// LS Electric XG5000 project: 커스텀통신시도1
// PLC LSPLC

PROGRAM NewProgram (task: 스캔 프로그램)

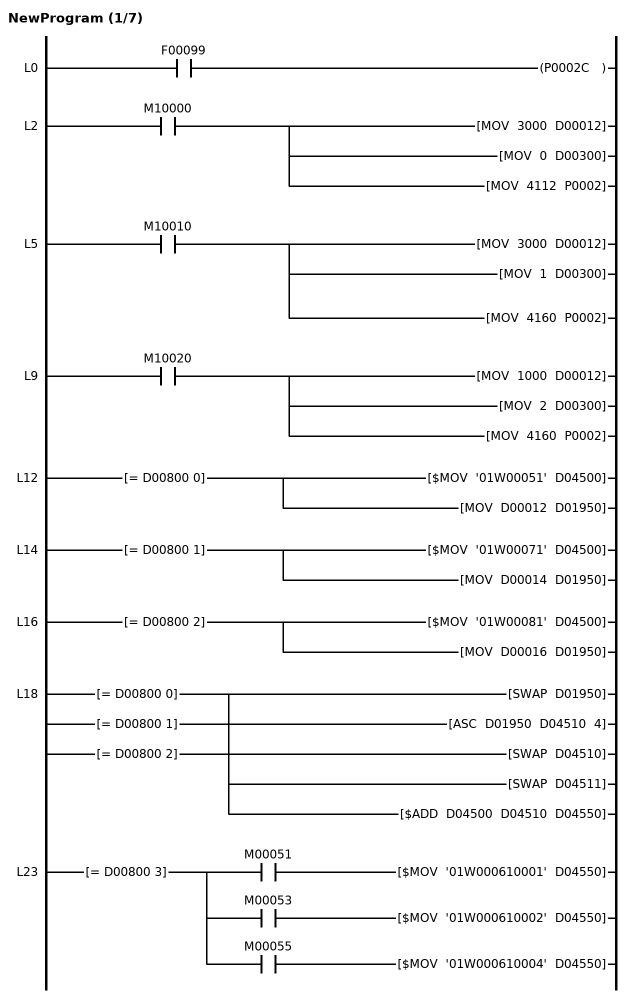
; L0
LOAD      F00099
OUT       P0002C
; L2
LOAD      M10000
MOV       3000 D00012
MOV       0 D00300
MOV       4112 P0002
; L5
LOAD      M10010
MOV       3000 D00012
MOV       1 D00300
MOV       4160 P0002
; L9
LOAD      M10020
MOV       1000 D00012
MOV       2 D00300
MOV       4160 P0002
; L12
LOAD=     D00800 0
$MOV      '01W00051' D04500
MOV       D00012 D01950
; L14
LOAD=     D00800 1
$MOV      '01W00071' D04500
MOV       D00014 D01950
; L16
LOAD=     D00800 2
$MOV      '01W00081' D04500
MOV       D00016 D01950
; L18
LOAD=     D00800 0
OR=       D00800 1
OR=       D00800 2
SWAP      D01950
ASC       D01950 D04510 4
SWAP      D04510
SWAP      D04511
$ADD      D04500 D04510 D04550
; L23
LOAD=     D00800 3
MPUSH
AND       M00051
$MOV      '01W000610001' D04550
MLOAD
AND       M00053
$MOV      '01W000610002' D04550
MPOP
AND       M00055
$MOV      '01W000610004' D04550

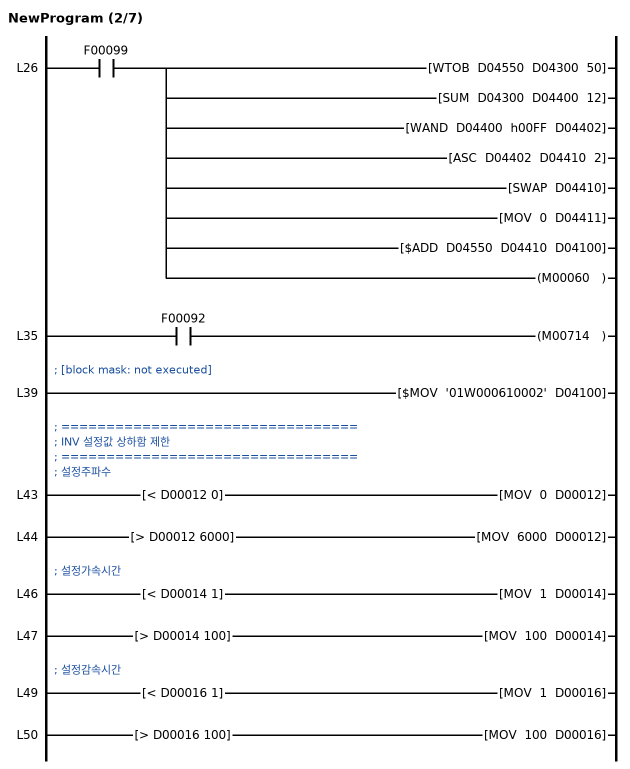
; L26
LOAD      F00099
WTOB      D04550 D04300 50
SUM       D04300 D04400 12
WAND      D04400 h00FF D04402
ASC       D04402 D04410 2
SWAP      D04410
MOV       0 D04411
$ADD      D04550 D04410 D04100
OUT       M00060
; L35
LOAD      F00092
OUT       M00714
; L39 (block mask: not executed)
$MOV      '01W000610002' D04100
// =================================
//    INV 설정값 상하함 제한
// =================================
// 설정주파수
; L43
LOAD<     D00012 0
MOV       0 D00012
; L44
LOAD>     D00012 6000
MOV       6000 D00012
// 설정가속시간
; L46
LOAD<     D00014 1
MOV       1 D00014
; L47
LOAD>     D00014 100
MOV       100 D00014
// 설정감속시간
; L49
LOAD<     D00016 1
MOV       1 D00016
; L50
LOAD>     D00016 100
MOV       100 D00016

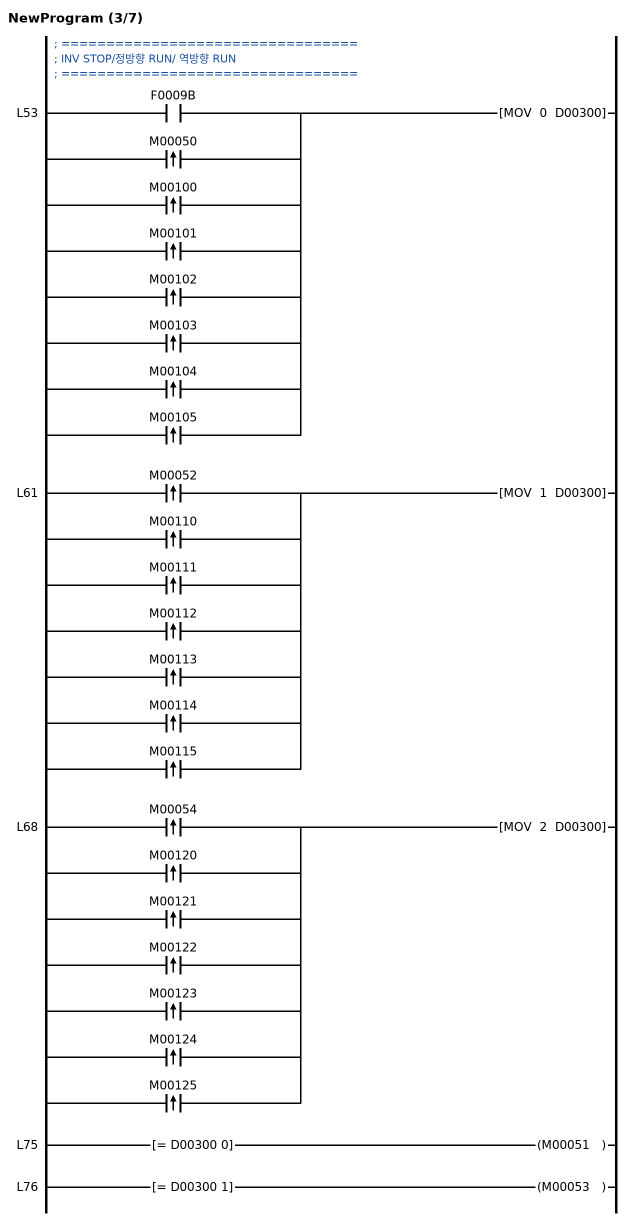
// =================================
//    INV STOP/정방향 RUN/ 역방향 RUN
// =================================
; L53
LOAD      F0009B
ORP       M00050
ORP       M00100
ORP       M00101
ORP       M00102
ORP       M00103
ORP       M00104
ORP       M00105
MOV       0 D00300
; L61
LOADP     M00052
ORP       M00110
ORP       M00111
ORP       M00112
ORP       M00113
ORP       M00114
ORP       M00115
MOV       1 D00300
; L68
LOADP     M00054
ORP       M00120
ORP       M00121
ORP       M00122
ORP       M00123
ORP       M00124
ORP       M00125
MOV       2 D00300
; L75
LOAD=     D00300 0
OUT       M00051
; L76
LOAD=     D00300 1
OUT       M00053

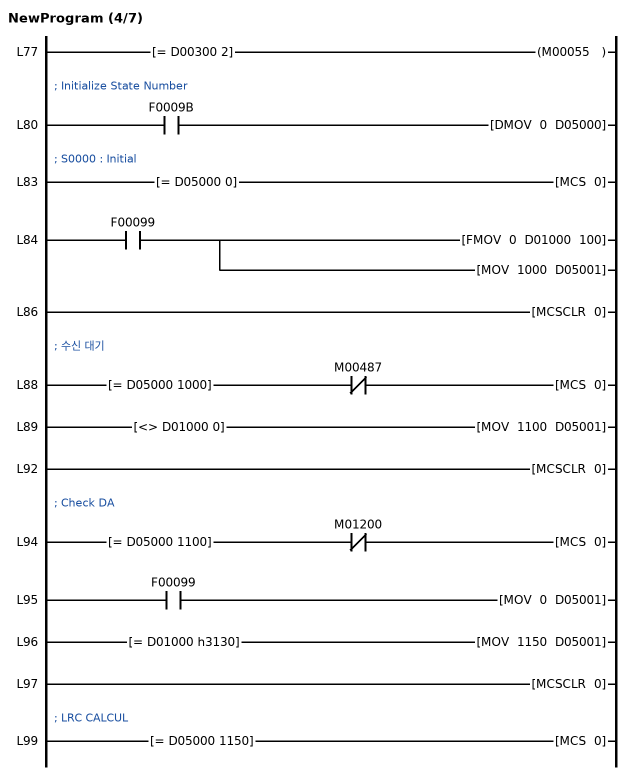
; L77
LOAD=     D00300 2
OUT       M00055
// Initialize State Number
; L80
LOAD      F0009B
DMOV      0 D05000
// S0000 : Initial
; L83
LOAD=     D05000 0
MCS       0
; L84
LOAD      F00099
FMOV      0 D01000 100
MOV       1000 D05001
; L86
MCSCLR    0
// 수신 대기
; L88
LOAD=     D05000 1000
AND NOT   M00487
MCS       0
; L89
LOAD<>    D01000 0
MOV       1100 D05001
; L92
MCSCLR    0
// Check DA
; L94
LOAD=     D05000 1100
AND NOT   M01200
MCS       0
; L95
LOAD      F00099
MOV       0 D05001
; L96
LOAD=     D01000 h3130
MOV       1150 D05001
; L97
MCSCLR    0
// LRC CALCUL
; L99
LOAD=     D05000 1150
MCS       0

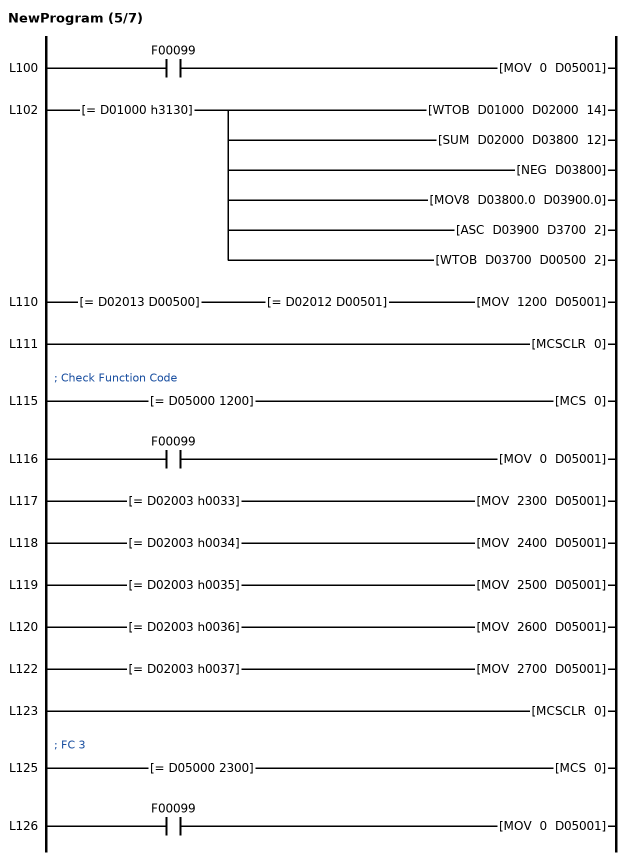
; L100
LOAD      F00099
MOV       0 D05001
; L102
LOAD=     D01000 h3130
WTOB      D01000 D02000 14
SUM       D02000 D03800 12
NEG       D03800
MOV8      D03800.0 D03900.0
ASC       D03900 D3700 2
WTOB      D03700 D00500 2
; L110
LOAD=     D02013 D00500
AND=      D02012 D00501
MOV       1200 D05001
; L111
MCSCLR    0
// Check Function Code
; L115
LOAD=     D05000 1200
MCS       0
; L116
LOAD      F00099
MOV       0 D05001
; L117
LOAD=     D02003 h0033
MOV       2300 D05001
; L118
LOAD=     D02003 h0034
MOV       2400 D05001
; L119
LOAD=     D02003 h0035
MOV       2500 D05001
; L120
LOAD=     D02003 h0036
MOV       2600 D05001
; L122
LOAD=     D02003 h0037
MOV       2700 D05001
; L123
MCSCLR    0
// FC 3
; L125
LOAD=     D05000 2300
MCS       0
; L126
LOAD      F00099
MOV       0 D05001

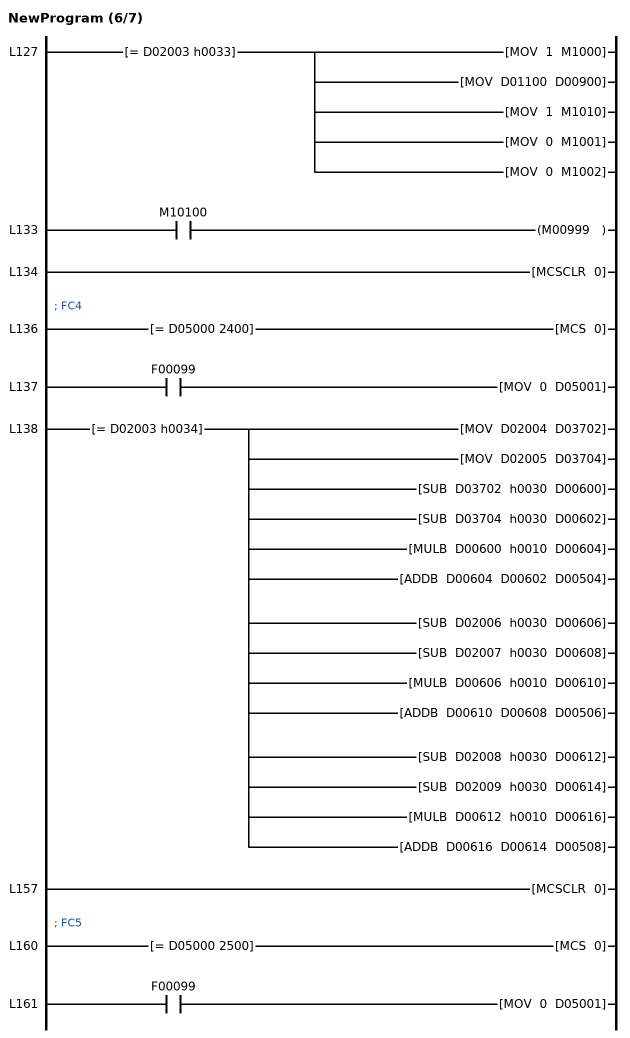
; L127
LOAD=     D02003 h0033
MOV       1 M1000
MOV       D01100 D00900
MOV       1 M1010
MOV       0 M1001
MOV       0 M1002
; L133
LOAD      M10100
OUT       M00999
; L134
MCSCLR    0
// FC4
; L136
LOAD=     D05000 2400
MCS       0
; L137
LOAD      F00099
MOV       0 D05001
; L138
LOAD=     D02003 h0034
MOV       D02004 D03702
MOV       D02005 D03704
SUB       D03702 h0030 D00600
SUB       D03704 h0030 D00602
MULB      D00600 h0010 D00604
ADDB      D00604 D00602 D00504
SUB       D02006 h0030 D00606
SUB       D02007 h0030 D00608
MULB      D00606 h0010 D00610
ADDB      D00610 D00608 D00506
SUB       D02008 h0030 D00612
SUB       D02009 h0030 D00614
MULB      D00612 h0010 D00616
ADDB      D00616 D00614 D00508
; L157
MCSCLR    0
// FC5
; L160
LOAD=     D05000 2500
MCS       0
; L161
LOAD      F00099
MOV       0 D05001

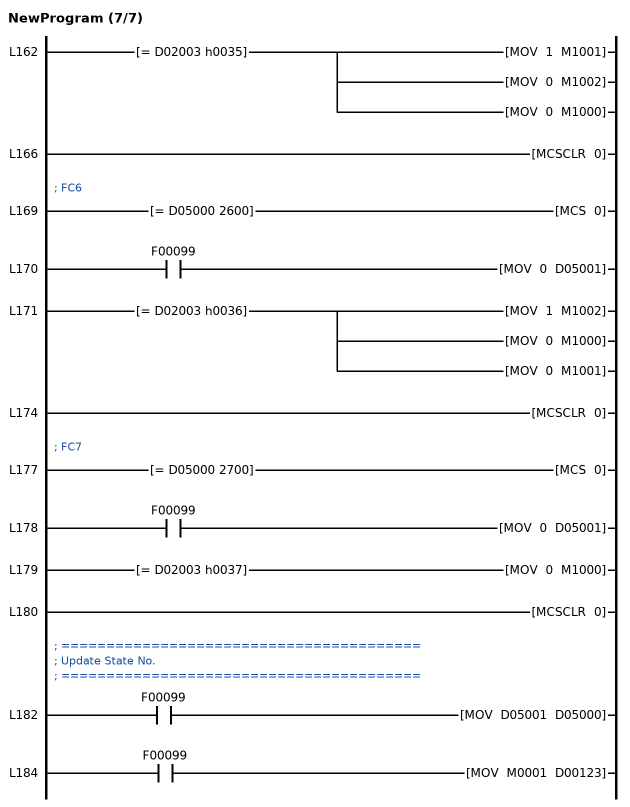
; L162
LOAD=     D02003 h0035
MOV       1 M1001
MOV       0 M1002
MOV       0 M1000
; L166
MCSCLR    0
// FC6
; L169
LOAD=     D05000 2600
MCS       0
; L170
LOAD      F00099
MOV       0 D05001
; L171
LOAD=     D02003 h0036
MOV       1 M1002
MOV       0 M1000
MOV       0 M1001
; L174
MCSCLR    0
// FC7
; L177
LOAD=     D05000 2700
MCS       0
; L178
LOAD      F00099
MOV       0 D05001
; L179
LOAD=     D02003 h0037
MOV       0 M1000
; L180
MCSCLR    0
// ========================================
// Update State No.
// ========================================
; L182
LOAD      F00099
MOV       D05001 D05000
; L184
LOAD      F00099
MOV       M0001 D00123